{attribute 'GeneratedUsingTerminal: EK1100-0000-0018'}
{attribute addProperty BoxType "EK1100-0000-0018"}
{attribute addProperty Id "R4A2_EK1122EK1122_1FC0878B2R4A3_EL1809EL1809_32157CFD20R4A4_EL1809EL1809_32157CFD20R4A5_EL1809EL1809_32157CFD20R4A6_EL1809EL1809_32157CFD20R4A8_EL2809EL2809_2B6483BD19R4A9_EL2809EL2809_2B6483BD19R4A10_EL1809EL1809_32157CFD20R4A11_EL2809EL2809_2B6483BD19"}
{attribute addProperty CRC "1904109275"}
{attribute addProperty Size "159"}
TYPE R4_EK1100_717E66DB EXTENDS EK1100_1FC0878B :
STRUCT
	{attribute addProperty Name "R4A2_EK1122"}
	{attribute addProperty PreviousPort "R4 (EK1100) : B"}
	R4A2_EK1122 : EK1122_1FC0878B;
	{attribute addProperty Name "R4A3_EL1809"}
	{attribute addProperty PreviousPort "R4A2 (EK1122) : C"}
	R4A3_EL1809 : EL1809_32157CFD;
	{attribute addProperty Name "R4A4_EL1809"}
	{attribute addProperty PreviousPort "R4A3 (EL1809) : B"}
	R4A4_EL1809 : EL1809_32157CFD;
	{attribute addProperty Name "R4A5_EL1809"}
	{attribute addProperty PreviousPort "R4A4 (EL1809) : B"}
	R4A5_EL1809 : EL1809_32157CFD;
	{attribute addProperty Name "R4A6_EL1809"}
	{attribute addProperty PreviousPort "R4A5 (EL1809) : B"}
	R4A6_EL1809 : EL1809_32157CFD;
	{attribute addProperty Name "R4A8_EL2809"}
	{attribute addProperty PreviousPort "R4A6 (EL1809) : B"}
	R4A8_EL2809 : EL2809_2B6483BD;
	{attribute addProperty Name "R4A9_EL2809"}
	{attribute addProperty PreviousPort "R4A8 (EL2809) : B"}
	R4A9_EL2809 : EL2809_2B6483BD;
	{attribute addProperty Name "R4A10_EL1809"}
	{attribute addProperty PreviousPort "R4A9 (EL2809) : B"}
	R4A10_EL1809 : EL1809_32157CFD;
	{attribute addProperty Name "R4A11_EL2809"}
	{attribute addProperty PreviousPort "R4A10 (EL1809) : B"}
	R4A11_EL2809 : EL2809_2B6483BD;
END_STRUCT
END_TYPE

(* stored: Version 1.2.0.0, ProductVersion 3.1.4024.9
   DUT R4_EK1100_717E66DB: Id {9c84d1c4-0420-0de1-04c8-8048a84ecd40} *)
